PROGRAM PG_Rain
VAR
	Regenmacher: FB_Regenmacher;;
	Wetterbericht: FB_Wetterbericht;
END_VAR
VAR // added by the converter: edge detectors and wires of the graphical bodies
    _w1 : ANY;
END_VAR

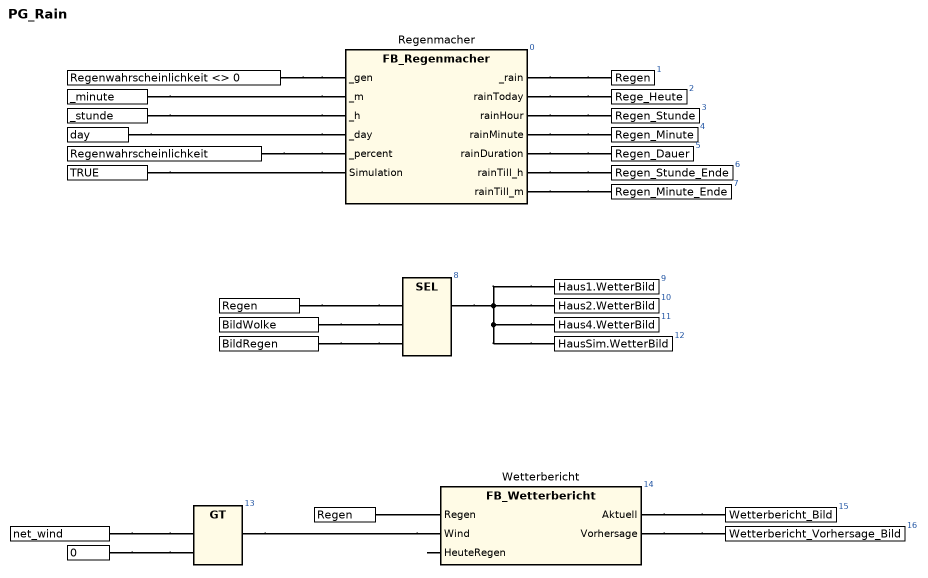
Regenmacher(
    _gen := Regenwahrscheinlichkeit <> 0,
    _m := _minute,
    _h := _stunde,
    _day := day,
    _percent := Regenwahrscheinlichkeit,
    Simulation := TRUE); // FB_Regenmacher
Regen := Regenmacher._rain;
Rege_Heute := Regenmacher.rainToday;
Regen_Stunde := Regenmacher.rainHour;
Regen_Minute := Regenmacher.rainMinute;
Regen_Dauer := Regenmacher.rainDuration;
Regen_Stunde_Ende := Regenmacher.rainTill_h;
Regen_Minute_Ende := Regenmacher.rainTill_m;
_w1 := SEL(Regen, BildWolke, BildRegen);
Haus1.WetterBild := _w1;
Haus2.WetterBild := _w1;
Haus4.WetterBild := _w1;
HausSim.WetterBild := _w1;
Wetterbericht(Regen := Regen, Wind := net_wind > 0); // FB_Wetterbericht
Wetterbericht_Bild := Wetterbericht.Aktuell;
Wetterbericht_Vorhersage_Bild := Wetterbericht.Vorhersage;

END_PROGRAM

(* stored: Version 1.1.0.1, ProductVersion 3.1.4018.5
   POU PG_Rain: Id {adb02757-c25f-4f7e-abb3-6e14f23bc446}, SpecialFunc None *)
